FUNCTION F_CoolTank 

VAR_INPUT
	refTank : REFERENCE TO ST_Tank;
END_VAR

IF refTank.temperature > 50 THEN
	refTank.temperature := refTank.temperature - 1;
END_IF

END_FUNCTION

(* stored: Version 1.1.0.1, ProductVersion 3.1.4024.16
   POU F_CoolTank: Id {93587bc4-3546-4283-bd19-cf03bd238455}, SpecialFunc None *)
